(* PLC project ST_traffic_light.project, CODESYS CODESYS V3.5 SP15 Patch 3 *)
(* stored: creationDateTime 2020-12-19T08:49:31.180402, modificationDateTime 2020-12-19T08:42:11.7060485 *)

PROGRAM POU
  VAR
    greenSec : WORD := 3;
    greenFlinkSec : WORD := 2;
    yellowSec : WORD := 2;
    redSec : WORD := 7;
    waitSec : WORD := greenSec;
    waitTimer : TON;
    flickTimer : TON;
    greenLight : BOOL := TRUE;
    yellowLight : BOOL := FALSE;
    redLight : BOOL := FALSE;
    nextStatus : INT := 1;
  END_VAR

            
waitTimer(IN := NOT waitTimer.Q, PT :=WORD_TO_TIME(waitSec * 1000));

IF waitTimer.Q = TRUE THEN
	CASE nextStatus OF
		0:  greenLight := TRUE;
			yellowLight := redLight := FALSE;
			waitSec := greenSec;
			nextStatus := 1;
		1:	waitSec := greenFlinkSec;
			nextStatus := 5;
		5:  yellowLight := TRUE;
			greenLight := redLight := FALSE;
			waitSec := yellowSec;
			nextStatus := 10;
		10:  redLight := TRUE;
			greenLight := yellowLight := FALSE;
			waitSec := redSec;
			nextStatus := 0;
	END_CASE	
END_IF

IF nextStatus = 5 THEN
	flickTimer(IN := NOT flickTimer.Q, PT := T#500MS);
	IF flickTimer.Q = TRUE THEN
		greenLight := NOT greenLight;
		//IF greenLight = TRUE THEN
		//	greenLight := FALSE;
		//ELSE
		//	greenLight := TRUE;
		//END_IF
	END_IF
END_IF	

          
END_PROGRAM
